// SIMATIC STEP 7 (V5.x) project bt4
// CPU: CPU 314C-2 DP
// station: Hardware
// station: SIMATIC 300(1)
// station: P_ADR_BUS
// program: S7 Program(1)

SYMBOL_TABLE
"START"	I 0.0	BOOL
"STOP"	I 0.1	BOOL
"A1"	I 0.2	BOOL
"A2"	I 0.3	BOOL
"B1"	I 0.4	BOOL
"B2"	I 0.5	BOOL
"D1"	I 0.6	BOOL
"D2"	I 0.7	BOOL
"E1"	I 1.0	BOOL
"E2"	I 1.1	BOOL
"G1"	I 1.2	BOOL
"G2"	I 1.3	BOOL
"H1"	I 1.4	BOOL
"H2"	I 1.5	BOOL
"YS"	M 0.0	BOOL
"Y1"	M 0.1	BOOL
"Y2"	M 0.2	BOOL
"Y3"	M 0.3	BOOL
"Y4"	M 0.4	BOOL
"Y5"	M 0.5	BOOL
"Y6"	M 0.6	BOOL
"Y7"	M 0.7	BOOL
"Y8"	M 1.0	BOOL
"Y9"	M 1.1	BOOL
"Y10"	M 1.2	BOOL
"Y11"	M 1.3	BOOL
"Y12"	M 1.4	BOOL
"Y13"	M 1.5	BOOL
"Y14"	M 1.6	BOOL
"CNT"	M 1.7	BOOL
"A"	Q 0.0	BOOL
"B"	Q 0.1	BOOL
"D"	Q 0.2	BOOL
"E"	Q 0.3	BOOL
"G"	Q 0.4	BOOL
"H"	Q 0.5	BOOL
END_SYMBOL_TABLE

ORGANIZATION_BLOCK OB 1
TITLE = "Main Program Sweep (Cycle)"
VERSION : 0.1
VAR_TEMP
  OB1_EV_CLASS : BYTE ;	//Bits 0-3 = 1 (Coming event), Bits 4-7 = 1 (Event class 1)
  OB1_SCAN_1 : BYTE ;	//1 (Cold restart scan 1 of OB 1), 3 (Scan 2-n of OB 1)
  OB1_PRIORITY : BYTE ;	//Priority of OB Execution
  OB1_OB_NUMBR : BYTE ;	//1 (Organization block 1, OB1)
  OB1_RESERVED_1 : BYTE ;	//Reserved for system
  OB1_RESERVED_2 : BYTE ;	//Reserved for system
  OB1_PREV_CYCLE : INT ;	//Cycle time of previous OB1 scan (milliseconds)
  OB1_MIN_CYCLE : INT ;	//Minimum cycle time of OB1 (milliseconds)
  OB1_MAX_CYCLE : INT ;	//Maximum cycle time of OB1 (milliseconds)
  OB1_DATE_TIME : DATE_AND_TIME ;	//Date and time OB1 started
END_VAR
BEGIN
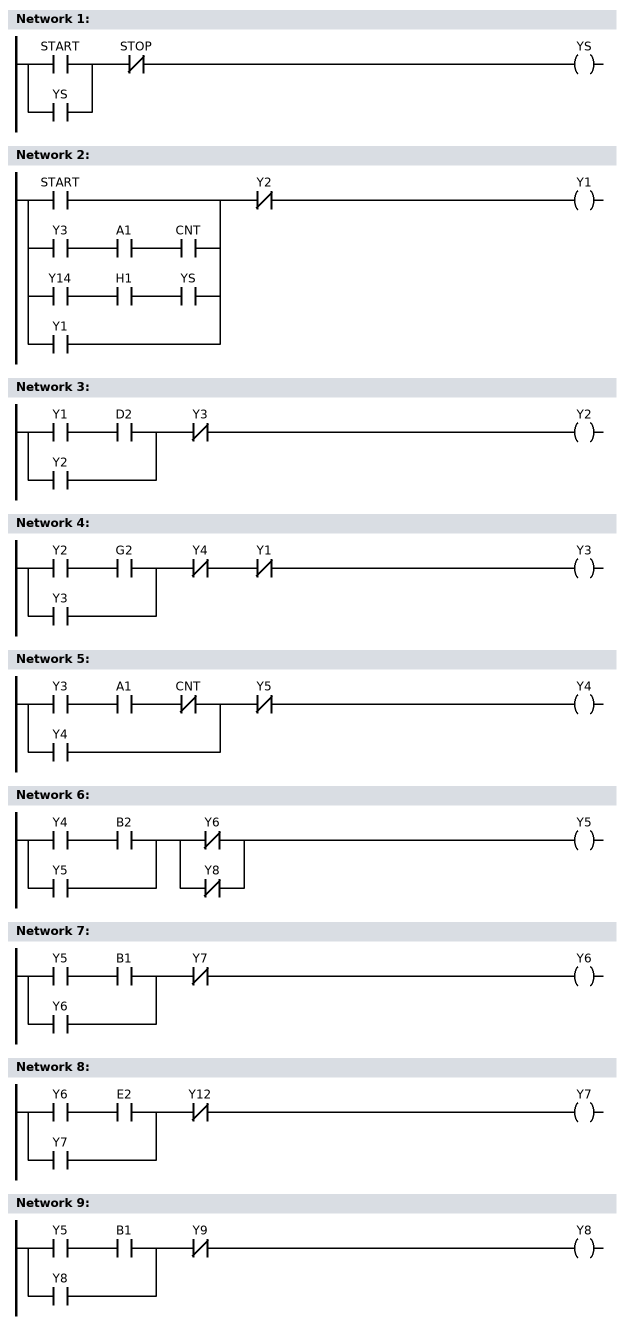
NETWORK
TITLE =
      A(;
      O     "START";
      O     "YS";
      );
      AN    "STOP";
      =     "YS";
NETWORK
TITLE =
      A(;
      O     "START";
      O;
      A     "Y3";
      A     "A1";
      A     "CNT";
      O;
      A     "Y14";
      A     "H1";
      A     "YS";
      O     "Y1";
      );
      AN    "Y2";
      =     "Y1";
NETWORK
TITLE =
      A(;
      A     "Y1";
      A     "D2";
      O     "Y2";
      );
      AN    "Y3";
      =     "Y2";
NETWORK
TITLE =
      A(;
      A     "Y2";
      A     "G2";
      O     "Y3";
      );
      AN    "Y4";
      AN    "Y1";
      =     "Y3";
NETWORK
TITLE =
      A(;
      A     "Y3";
      A     "A1";
      AN    "CNT";
      O     "Y4";
      );
      AN    "Y5";
      =     "Y4";
NETWORK
TITLE =
      A(;
      A     "Y4";
      A     "B2";
      O     "Y5";
      );
      A(;
      ON    "Y6";
      ON    "Y8";
      );
      =     "Y5";
NETWORK
TITLE =
      A(;
      A     "Y5";
      A     "B1";
      O     "Y6";
      );
      AN    "Y7";
      =     "Y6";
NETWORK
TITLE =
      A(;
      A     "Y6";
      A     "E2";
      O     "Y7";
      );
      AN    "Y12";
      =     "Y7";
NETWORK
TITLE =
      A(;
      A     "Y5";
      A     "B1";
      O     "Y8";
      );
      AN    "Y9";
      =     "Y8";
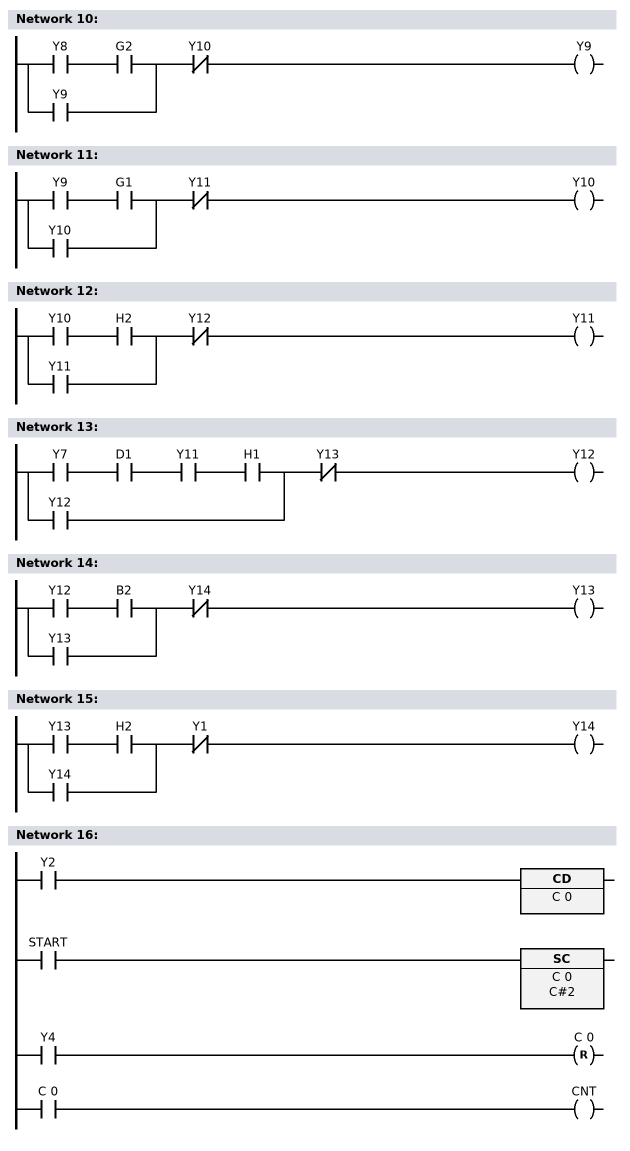
NETWORK
TITLE =
      A(;
      A     "Y8";
      A     "G2";
      O     "Y9";
      );
      AN    "Y10";
      =     "Y9";
NETWORK
TITLE =
      A(;
      A     "Y9";
      A     "G1";
      O     "Y10";
      );
      AN    "Y11";
      =     "Y10";
NETWORK
TITLE =
      A(;
      A     "Y10";
      A     "H2";
      O     "Y11";
      );
      AN    "Y12";
      =     "Y11";
NETWORK
TITLE =
      A(;
      A     "Y7";
      A     "D1";
      A     "Y11";
      A     "H1";
      O     "Y12";
      );
      AN    "Y13";
      =     "Y12";
NETWORK
TITLE =
      A(;
      A     "Y12";
      A     "B2";
      O     "Y13";
      );
      AN    "Y14";
      =     "Y13";
NETWORK
TITLE =
      A(;
      A     "Y13";
      A     "H2";
      O     "Y14";
      );
      AN    "Y1";
      =     "Y14";
NETWORK
TITLE =
      A     "Y2";
      CD    C 0;
      BLD   101;
      A     "START";
      L     C#2;
      S     C 0;
      A     "Y4";
      R     C 0;
      NOP   0;
      NOP   0;
      A     C 0;
      =     "CNT";
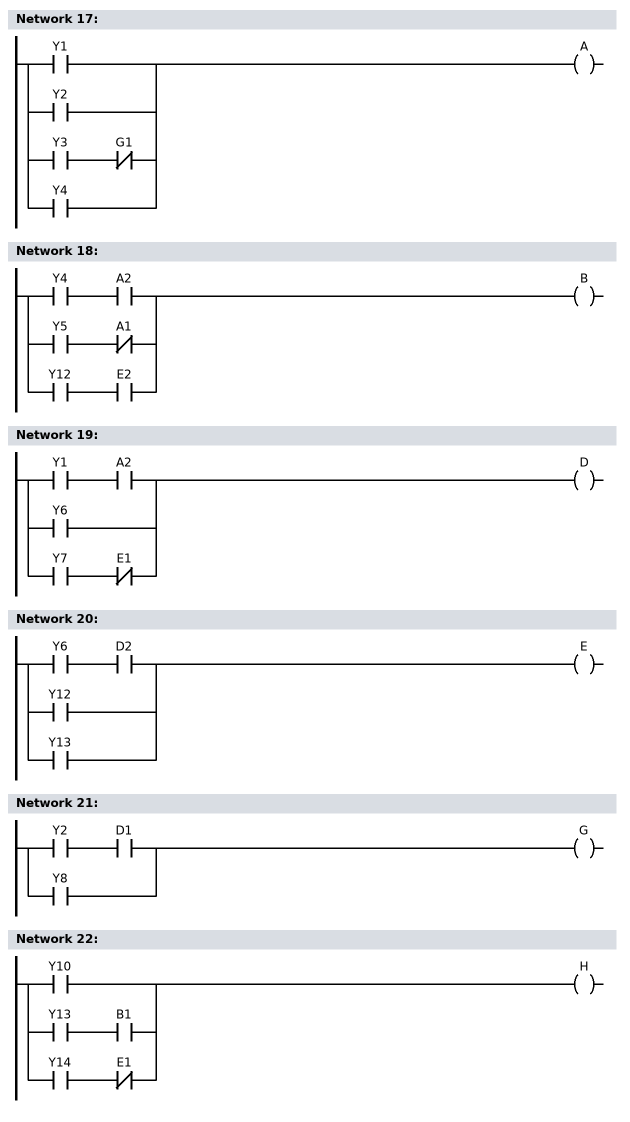
NETWORK
TITLE =
      O     "Y1";
      O     "Y2";
      O;
      A     "Y3";
      AN    "G1";
      O     "Y4";
      =     "A";
NETWORK
TITLE =
      A     "Y4";
      A     "A2";
      O;
      A     "Y5";
      AN    "A1";
      O;
      A     "Y12";
      A     "E2";
      =     "B";
NETWORK
TITLE =
      A     "Y1";
      A     "A2";
      O     "Y6";
      O;
      A     "Y7";
      AN    "E1";
      =     "D";
NETWORK
TITLE =
      A     "Y6";
      A     "D2";
      O     "Y12";
      O     "Y13";
      =     "E";
NETWORK
TITLE =
      A     "Y2";
      A     "D1";
      O     "Y8";
      =     "G";
NETWORK
TITLE =
      O     "Y10";
      O;
      A     "Y13";
      A     "B1";
      O;
      A     "Y14";
      AN    "E1";
      =     "H";
END_ORGANIZATION_BLOCK
